RoboDK station: virtual_scene.rdk

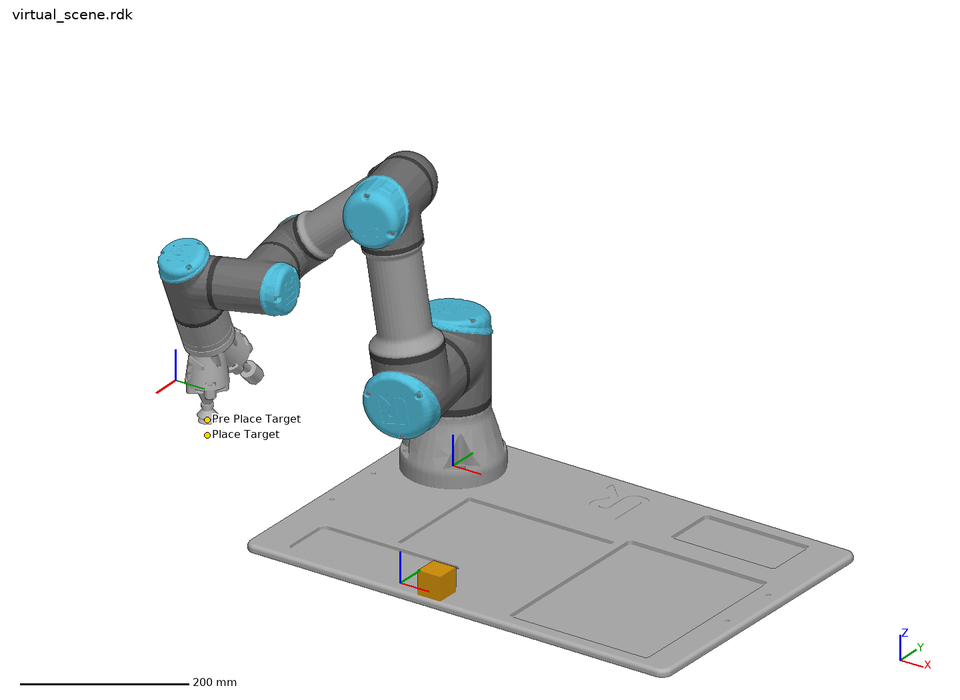
[picture v0: the station drawn from its stored meshes, robots at their saved joint values, targets as dots, program paths as lines]
Station virtual_scene (saved by RoboDK 5.9.0). Poses are relative to the parent item; angles as X-Y-Z fixed-axis rotations.
Station parameters (name, value as stored): LIN64
  - frame UR3e Base at (0, 0, 0) mm
    - robot UR3e: 6 axes, payload 3 kg, reach 500 mm, repeatability 0.03 mm, weight 11 kg
        modified DH rows (alpha deg, a mm, theta deg, d mm): 0, 0, 0, 151.9; 90, 0, 180, 0; 0, 243.55, 0, 0; 0, 213.2, 0, 131.05; -90, 0, 0, 85.35; 90, 0, 180, 92.1
        joint limits [-360, -360, -360, -360, -360, -360] to [360, 360, 360, 360, 360, 360]; home [0, -90, 0, -90, 0, 0]; saved at [11.776, -81.963, 121.841, -124.926, -112.489, 12.761]
      - tool HerramientaDual_borr, TCP at (-44.63, 0, 105.14) mm, rotated rx 0 ry -23 rz 0 deg, size 118.6 x 63 x 135.8 mm
    - object BaseRobotUR3e at (525, 85, -10) mm, rotated rx 0 ry 0 rz 180 deg, size 610 x 398 x 10 mm, geometry from BaseRobotUR3e.STL
  - frame World Frame at (130.34, -294.32, 0) mm
    - object Item 1 at (50, 0, 0) mm, size 32.5 x 32.5 x 32.5 mm, geometry from Cube-500mm.sld
  - Python program Main Program (listed below)
  - frame Place Frame at (-400, 0, 0) mm, rotated rx 0 ry 0 rz -90 deg
    - target Pre Place Target (Cartesian target) at (150, 150, 50) mm, rotated rx 180 ry 0 rz -180 deg; joints [11.776, -81.963, 121.841, -124.926, -112.489, 12.761] of UR3e
    - target Place Target (Cartesian target) at (150, 150, 30) mm, rotated rx 180 ry 0 rz -180 deg; joints [11.776, -78.13, 124.329, -131.248, -112.489, 12.761] of UR3e

--- Python program Main Program ---
# Type help("robodk.robolink") or help("robodk.robomath") for more information
# Press F5 to run the script
# Documentation: https://robodk.com/doc/en/RoboDK-API.html
# Reference:     https://robodk.com/doc/en/PythonAPI/robodk.html
# Note: It is not required to keep a copy of this file, your Python script is saved with your RDK project


# ---------------------------------------------------------------------------- #
# IMPORTACIONES NECESARIAS

from json.__init__ import loads as json_loads
import paho.mqtt.client as mqtt
import numpy as np

from robodk import robolink    # RoboDK API
from robodk import robomath    # Robot toolbox

from robodk.robolink import ITEM_TYPE_OBJECT
from robodk.robomath import TxyzRxyz_2_Pose

RDK = robolink.Robolink()
item_01 = RDK.Item('Item 1', ITEM_TYPE_OBJECT)
robot = RDK.Item('UR3e')
tool = RDK.Item('HerramientaDual_borr')

# Establecer herramienta de la herramienta industria:
robot.setTool(tool)

# ---------------------------------------------------------------------------- #
# PARÁMETROS Y TOPICS PARA LA CONEXIÓN CON MQTT

BROKER   = 'broker.emqx.io'
PORT     =  1883
USERNAME = 'emqx'
PASSWORD = 'public'

POSITION_TOPIC = "robodk/position"


# ---------------------------------------------------------------------------- #
# FUNCIONES DESARROLLADAS

def on_message(mqttc, obj, msg):
    """
    Función que analiza el topic recibido y realiza la acción oportuna.
    """

    # El primer paso es parsear msg:
    msg_dict = json_loads((msg.payload).decode('UTF-8'))

    if msg.topic == POSITION_TOPIC:
        new_pose = TxyzRxyz_2_Pose(
            [msg_dict["x"] * 10.0,
	     msg_dict["y"] * 10.0,
	     msg_dict["z"] * 10.0,
	     0.0, 0.0, 0.0])

        item_01.setPose(new_pose)

        pre_pick_pose = TxyzRxyz_2_Pose(
            [msg_dict["x"] * 10.0,
	     msg_dict["y"] * 10.0,
	     (msg_dict["z"] + 10) * 10.0,
	     0.0, np.pi, 0.0])

        pick_pose = TxyzRxyz_2_Pose(
            [msg_dict["x"] * 10.0,
	     msg_dict["y"] * 10.0,
	     (msg_dict["z"] + 3) * 10.0,
	     0.0, np.pi, 0.0])

        for i in range(1, msg_dict["quantity"] + 1):
            robot.setPoseFrame(RDK.Item('World Frame'))
            robot.MoveJ(pre_pick_pose, True)
            robot.MoveL(pick_pose, True)
            robot.MoveL(pre_pick_pose, True)

            robot.setPoseFrame(RDK.Item('Place Frame'))
            robot.MoveJ(RDK.Item('Pre Place Target'), True)
            robot.MoveL(RDK.Item('Place Target'), True)
            robot.MoveL(RDK.Item('Pre Place Target'), True)

# ---------------------------------------------------------------------------- #
# CREAR CLIENTE Y ESTABLECER CONEXIÓN MQTT (BUCLE)

client = mqtt.Client()
client.on_message = on_message

client.username_pw_set(username = USERNAME, password = PASSWORD)
client.connect(BROKER, PORT, 60)

client.subscribe(POSITION_TOPIC, 0)

client.loop_forever()

### end of file ###
